PROGRAM pouS2Prompts
VAR
	


idbMsgPrompt: FB_CheckMessageBounds;
END_VAR

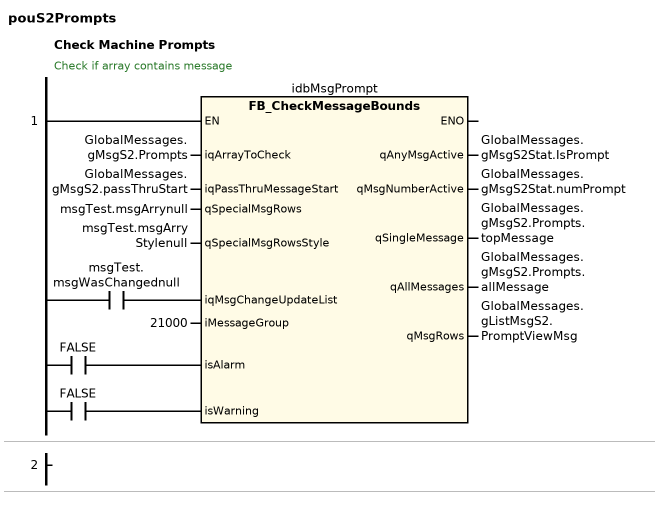
// NETWORK 1: Check Machine Prompts
// Check if array contains message
idbMsgPrompt(
    iqArrayToCheck := GlobalMessages.gMsgS2.Prompts,
    iqPassThruMessageStart := GlobalMessages.gMsgS2.passThruStart,
    qSpecialMsgRows := msgTest.msgArrynull,
    qSpecialMsgRowsStyle := msgTest.msgArryStylenull,
    iqMsgChangeUpdateList := msgTest.msgWasChangednull,
    iMessageGroup := 21000,
    isAlarm := FALSE,
    isWarning := FALSE,
    qAnyMsgActive => GlobalMessages.gMsgS2Stat.IsPrompt,
    qMsgNumberActive => GlobalMessages.gMsgS2Stat.numPrompt,
    qSingleMessage => GlobalMessages.gMsgS2.Prompts.topMessage,
    qAllMessages => GlobalMessages.gMsgS2.Prompts.allMessage,
    qMsgRows => GlobalMessages.gListMsgS2.PromptViewMsg); // FB_CheckMessageBounds

// NETWORK 2

END_PROGRAM

(* stored: Version 1.1.0.1, ProductVersion 3.1.4024.12
   POU pouS2Prompts: Id {27e7d3ad-8739-4cbe-a913-ad9edc9d3370}, SpecialFunc None *)
